// TIA Portal V17 export
// export: Created 2022-07-28T18:02:45.4276913Z, ExportSetting None, DisplayName Totally Integrated Automation Portal, DisplayVersion V17, DisplayName TIA Portal Openness, DisplayVersion V17, DisplayName TIA Portal Teamcenter Gateway, DisplayVersion V17, DisplayName TIA Portal Version Control Interface, DisplayVersion V17, DisplayName TIA Portal Test Suite Advanced, DisplayVersion V17, DisplayName SINAMICS Startdrive Advanced, DisplayVersion V17, DisplayName SINAMICS DCC, DisplayVersion V17, DisplayName SINAMICS Startdrive G130, G150, S120, S150, SINAMICS MV, S210, DisplayVersion V17, DisplayName SINAMICS Startdrive G110M, G120, G120C, G120D, G120P, G115D, DisplayVersion V17, DisplayName STEP 7 Professional, DisplayVersion V17, DisplayName SIMATIC Energy Suite, DisplayVersion V17, DisplayName STEP 7 CFC, DisplayVersion V17, DisplayName STEP 7 Safety, DisplayVersion V17, DisplayName WinCC Advanced / Unified PC, DisplayVersion V17, DisplayName SIMATIC Visualization Architect, DisplayVersion V17
FUNCTION "Lib_FC_GenMoto_InitInternal" : Void   // FC13, SCL
{ S7_Optimized_Access := 'TRUE' }
// stored: SetENOAutomatically false
   VAR_IN_OUT
      IQ_InternalData : "Lib_UDT_Int";   // Internal data
   END_VAR
BEGIN
   //Set internal data
   #IQ_InternalData.AlwTrue := true;
   #IQ_InternalData.AlwFalse := false;
   #IQ_InternalData.i_Alw0 := 0;
   #IQ_InternalData.b_Alw0 := b#16#0;
   #IQ_InternalData.w_Alw0 := w#16#0;
   #IQ_InternalData.d_Alw0 := dw#16#0;
END_FUNCTION
